FUNCTION_BLOCK FB_ConveyorMachine
VAR
	StopButton 				: I_Pushbutton;
	EmergencyStopButton 	: I_Pushbutton;
	StartButton 			: I_Pushbutton;
	ProductDetectedSensor 	: I_Sensor;
	ConveyorFullSensor		: I_Sensor;
	MotorContactor 			: FB_MotorContactor;
	Timeout 				: TOF;
	ConveyorControl 		: BOOL;
END_VAR

IF StopButton.IsPressed OR EmergencyStopButton.IsPressed THEN	
	ConveyorControl := FALSE;	
ELSIF StartButton.IsPressed AND StopButton.IsReleased AND EmergencyStopButton.IsReleased THEN
	ConveyorControl := TRUE;	
END_IF

Timeout(IN:= ConveyorControl AND ProductDetectedSensor.IsActive, PT:= T#5S);

IF ConveyorControl AND Timeout.Q AND NOT ConveyorFullSensor.IsActive THEN
	MotorContactor.SwitchOn();
ELSE
	MotorContactor.SwitchOff();
END_IF

METHOD FB_init : BOOL
VAR_INPUT
	bInitRetains : BOOL; // if TRUE, the retain variables are initialized (warm start / cold start)
	bInCopyCode : BOOL;  // if TRUE, the instance afterwards gets moved into the copy code (online change)
	StopButton 				: I_Pushbutton;
	EmergencyStopButton 	: I_Pushbutton;
	StartButton 			: I_Pushbutton;
	ProductDetectedSensor 	: I_Sensor;
	ConveyorFullSensor		: I_Sensor;
	MotorContactor 			: FB_MotorContactor;
END_VAR
THIS^.StopButton 				:= StopButton 			;
THIS^.EmergencyStopButton 		:= EmergencyStopButton 	;
THIS^.StartButton 				:= StartButton 			;
THIS^.ProductDetectedSensor 	:= ProductDetectedSensor;
THIS^.ConveyorFullSensor		:= ConveyorFullSensor	;
THIS^.MotorContactor 			:= MotorContactor 		;
END_METHOD

END_FUNCTION_BLOCK

(* stored: Version 1.1.0.1, ProductVersion 3.1.4024.13
   POU FB_ConveyorMachine: Id {bf8f32c4-ae24-4d88-8fd9-c5b105056ce8}, SpecialFunc None
   Method FB_init: Id {6da2375f-c1a0-4ca6-a605-6d38d414b673} *)
